# EPICS autosave request: ez4axis_example/as/req/all_motor_settings.req
file "motor_settings.req", P=$(P), M=m1
file "motor_settings.req", P=$(P), M=m2
file "motor_settings.req", P=$(P), M=m3
file "motor_settings.req", P=$(P), M=m4
